TYPE "LubrPump_Par"
VERSION : 0.1
// Block: LubrPump_Par
   STRUCT
      LowLevelCheckTime : Time;
      ValveONTime : Time;
      ValveOFFTime : Time;
   END_STRUCT;

END_TYPE
